// TIA Portal V17 export
// export: Created 2024-08-29T18:23:42.9804485Z, ExportSetting WithDefaults, DisplayName Totally Integrated Automation Portal, DisplayVersion V17 Update 7, DisplayName TIA Portal Openness, DisplayVersion V17 Update 7, DisplayName TIA Portal Version Control Interface, DisplayVersion V17, DisplayName SINAMICS Startdrive Advanced, DisplayVersion V17 SP2, DisplayName SINAMICS Startdrive G110M, G120, G120C, G120D, G120P, G115D, DisplayVersion V17 SP2, DisplayName SINAMICS Startdrive G130, G150, S120, S150, SINAMICS MV, S210, DisplayVersion V17 SP2, DisplayName STEP 7 Professional, DisplayVersion V17 Update 7, DisplayName STEP 7 Safety, DisplayVersion V17 Update 6, DisplayName WinCC Advanced / Unified PC, DisplayVersion V17 Update 7
FUNCTION "outputsMapping" : Void   // FC8, LAD
{ S7_Optimized_Access := 'TRUE' }
VERSION : 0.1
// stored: AutoNumber true, IsIECCheckEnabled false, SetENOAutomatically false, UDAEnableTagReadback false
BEGIN

REGION Network 1: STATION AIR ACTIVATION
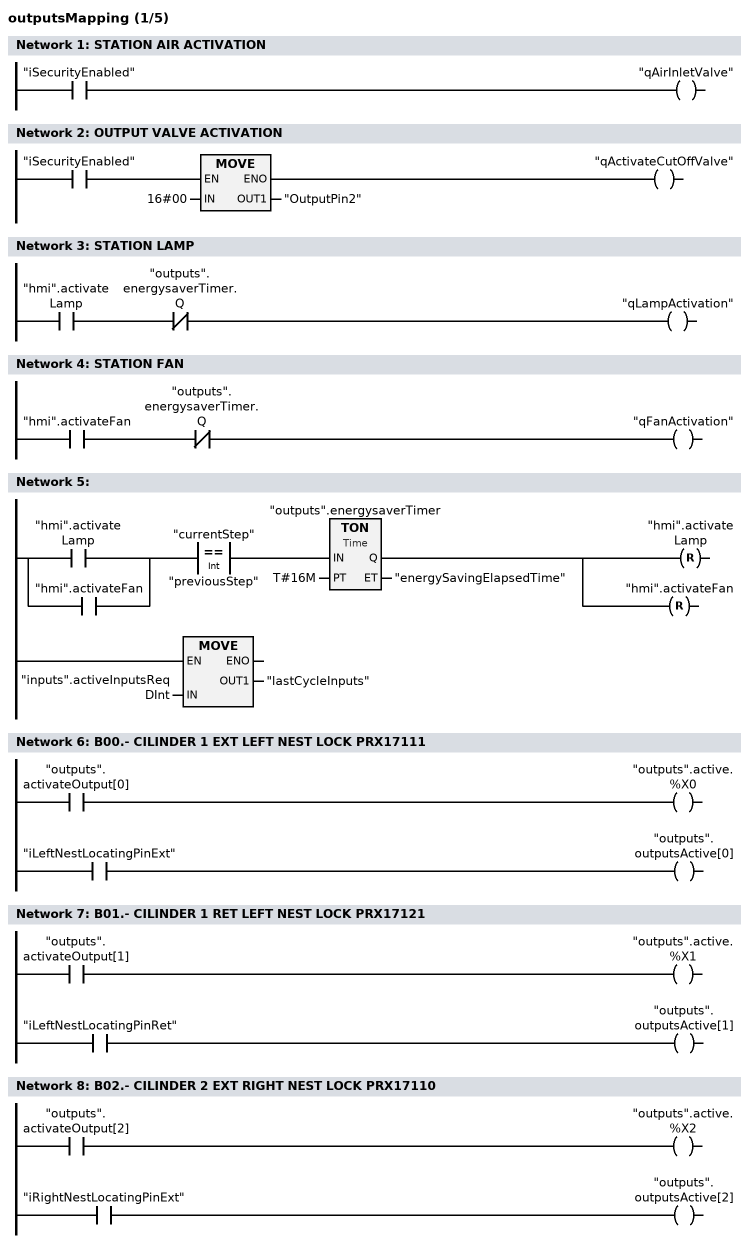
   RUNG wire#powerrail
      Contact( "iSecurityEnabled" )
      Coil( "qAirInletValve" )
   END_RUNG
   // the same network as SCL:
   "qAirInletValve" := "iSecurityEnabled";
END_REGION

REGION Network 2: OUTPUT VALVE ACTIVATION
   RUNG wire#powerrail
      Contact( "iSecurityEnabled" )
      Move(in := 16#00, out1 => "OutputPin2")
      Coil( "qActivateCutOffValve" )
   END_RUNG
   // the same network as SCL:
   IF "iSecurityEnabled" THEN "OutputPin2" := 16#00; END_IF;
   "qActivateCutOffValve" := "iSecurityEnabled";
END_REGION

REGION Network 3: STATION LAMP
   RUNG wire#powerrail
      Contact( "hmi".activateLamp )
      I_Contact( "outputs".energysaverTimer.Q )
      Coil( "qLampActivation" )
   END_RUNG
   // the same network as SCL:
   "qLampActivation" := "hmi".activateLamp AND NOT "outputs".energysaverTimer.Q;
END_REGION

REGION Network 4: STATION FAN
   RUNG wire#powerrail
      Contact( "hmi".activateFan )
      I_Contact( "outputs".energysaverTimer.Q )
      Coil( "qFanActivation" )
   END_RUNG
   // the same network as SCL:
   "qFanActivation" := "hmi".activateFan AND NOT "outputs".energysaverTimer.Q;
END_REGION

REGION Network 5
   RUNG wire#powerrail
      Contact( "hmi".activateLamp )
      wire#w1
      { S7_Templates := "SrcType := Int" } EQ_Contact(in1 := "currentStep", in2 := "previousStep")
      { S7_Templates := "time_type := Time" } "outputs".energysaverTimer.TON(pt := T#16M, et => "energySavingElapsedTime")
      wire#w2
      R_Coil( "hmi".activateLamp )
   END_RUNG
   RUNG wire#powerrail
      Contact( "hmi".activateFan )
   END_RUNG wire#w1
   RUNG wire#w2
      R_Coil( "hmi".activateFan )
   END_RUNG
   RUNG wire#powerrail
      Move(in := "inputs".activeInputsReqDInt, out1 => "lastCycleInputs")
   END_RUNG
   // the same network as SCL:
   "outputs".energysaverTimer.TON(IN := ("hmi".activateLamp OR "hmi".activateFan) AND ("currentStep" = "previousStep"),
                           PT := T#16M,
                           ET => "energySavingElapsedTime");
   IF "outputs".energysaverTimer.Q THEN
       "hmi".activateLamp := FALSE;
       "hmi".activateFan := FALSE;
   END_IF;
   "lastCycleInputs" := "inputs".activeInputsReqDInt;
END_REGION

REGION Network 6: B00.- CILINDER 1 EXT LEFT NEST LOCK PRX17111
   RUNG wire#powerrail
      Contact( "outputs".activateOutput[0] )
      Coil( "outputs".active.%X0 )
   END_RUNG
   RUNG wire#powerrail
      Contact( "iLeftNestLocatingPinExt" )
      Coil( "outputs".outputsActive[0] )
   END_RUNG
   // the same network as SCL:
   "outputs".active.%X0 := "outputs".activateOutput[0];
   "outputs".outputsActive[0] := "iLeftNestLocatingPinExt";
END_REGION

REGION Network 7: B01.- CILINDER 1 RET LEFT NEST LOCK PRX17121
   RUNG wire#powerrail
      Contact( "outputs".activateOutput[1] )
      Coil( "outputs".active.%X1 )
   END_RUNG
   RUNG wire#powerrail
      Contact( "iLeftNestLocatingPinRet" )
      Coil( "outputs".outputsActive[1] )
   END_RUNG
   // the same network as SCL:
   "outputs".active.%X1 := "outputs".activateOutput[1];
   "outputs".outputsActive[1] := "iLeftNestLocatingPinRet";
END_REGION

REGION Network 8: B02.- CILINDER 2 EXT RIGHT NEST LOCK PRX17110
   RUNG wire#powerrail
      Contact( "outputs".activateOutput[2] )
      Coil( "outputs".active.%X2 )
   END_RUNG
   RUNG wire#powerrail
      Contact( "iRightNestLocatingPinExt" )
      Coil( "outputs".outputsActive[2] )
   END_RUNG
   // the same network as SCL:
   "outputs".active.%X2 := "outputs".activateOutput[2];
   "outputs".outputsActive[2] := "iRightNestLocatingPinExt";
END_REGION

REGION Network 9: B03.- CILINDER 2 RET RIGHT NEST LOCK PRX17120
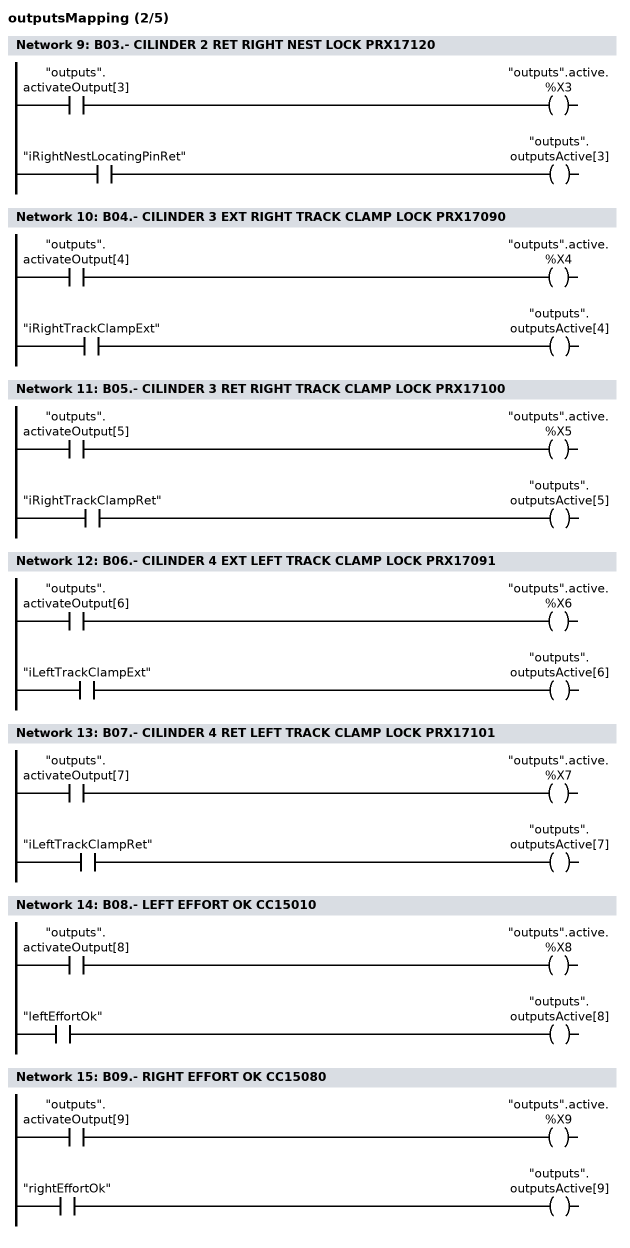
   RUNG wire#powerrail
      Contact( "outputs".activateOutput[3] )
      Coil( "outputs".active.%X3 )
   END_RUNG
   RUNG wire#powerrail
      Contact( "iRightNestLocatingPinRet" )
      Coil( "outputs".outputsActive[3] )
   END_RUNG
   // the same network as SCL:
   "outputs".active.%X3 := "outputs".activateOutput[3];
   "outputs".outputsActive[3] := "iRightNestLocatingPinRet";
END_REGION

REGION Network 10: B04.- CILINDER 3 EXT RIGHT TRACK CLAMP LOCK PRX17090
   RUNG wire#powerrail
      Contact( "outputs".activateOutput[4] )
      Coil( "outputs".active.%X4 )
   END_RUNG
   RUNG wire#powerrail
      Contact( "iRightTrackClampExt" )
      Coil( "outputs".outputsActive[4] )
   END_RUNG
   // the same network as SCL:
   "outputs".active.%X4 := "outputs".activateOutput[4];
   "outputs".outputsActive[4] := "iRightTrackClampExt";
END_REGION

REGION Network 11: B05.- CILINDER 3 RET RIGHT TRACK CLAMP LOCK PRX17100
   RUNG wire#powerrail
      Contact( "outputs".activateOutput[5] )
      Coil( "outputs".active.%X5 )
   END_RUNG
   RUNG wire#powerrail
      Contact( "iRightTrackClampRet" )
      Coil( "outputs".outputsActive[5] )
   END_RUNG
   // the same network as SCL:
   "outputs".active.%X5 := "outputs".activateOutput[5];
   "outputs".outputsActive[5] := "iRightTrackClampRet";
END_REGION

REGION Network 12: B06.- CILINDER 4 EXT LEFT TRACK CLAMP LOCK PRX17091
   RUNG wire#powerrail
      Contact( "outputs".activateOutput[6] )
      Coil( "outputs".active.%X6 )
   END_RUNG
   RUNG wire#powerrail
      Contact( "iLeftTrackClampExt" )
      Coil( "outputs".outputsActive[6] )
   END_RUNG
   // the same network as SCL:
   "outputs".active.%X6 := "outputs".activateOutput[6];
   "outputs".outputsActive[6] := "iLeftTrackClampExt";
END_REGION

REGION Network 13: B07.- CILINDER 4 RET LEFT TRACK CLAMP LOCK PRX17101
   RUNG wire#powerrail
      Contact( "outputs".activateOutput[7] )
      Coil( "outputs".active.%X7 )
   END_RUNG
   RUNG wire#powerrail
      Contact( "iLeftTrackClampRet" )
      Coil( "outputs".outputsActive[7] )
   END_RUNG
   // the same network as SCL:
   "outputs".active.%X7 := "outputs".activateOutput[7];
   "outputs".outputsActive[7] := "iLeftTrackClampRet";
END_REGION

REGION Network 14: B08.- LEFT EFFORT OK CC15010
   RUNG wire#powerrail
      Contact( "outputs".activateOutput[8] )
      Coil( "outputs".active.%X8 )
   END_RUNG
   RUNG wire#powerrail
      Contact( "leftEffortOk" )
      Coil( "outputs".outputsActive[8] )
   END_RUNG
   // the same network as SCL:
   "outputs".active.%X8 := "outputs".activateOutput[8];
   "outputs".outputsActive[8] := "leftEffortOk";
END_REGION

REGION Network 15: B09.- RIGHT EFFORT OK CC15080
   RUNG wire#powerrail
      Contact( "outputs".activateOutput[9] )
      Coil( "outputs".active.%X9 )
   END_RUNG
   RUNG wire#powerrail
      Contact( "rightEffortOk" )
      Coil( "outputs".outputsActive[9] )
   END_RUNG
   // the same network as SCL:
   "outputs".active.%X9 := "outputs".activateOutput[9];
   "outputs".outputsActive[9] := "rightEffortOk";
END_REGION

REGION Network 16: B10.- LEFT INSERTION OK DISTANCE SD14160
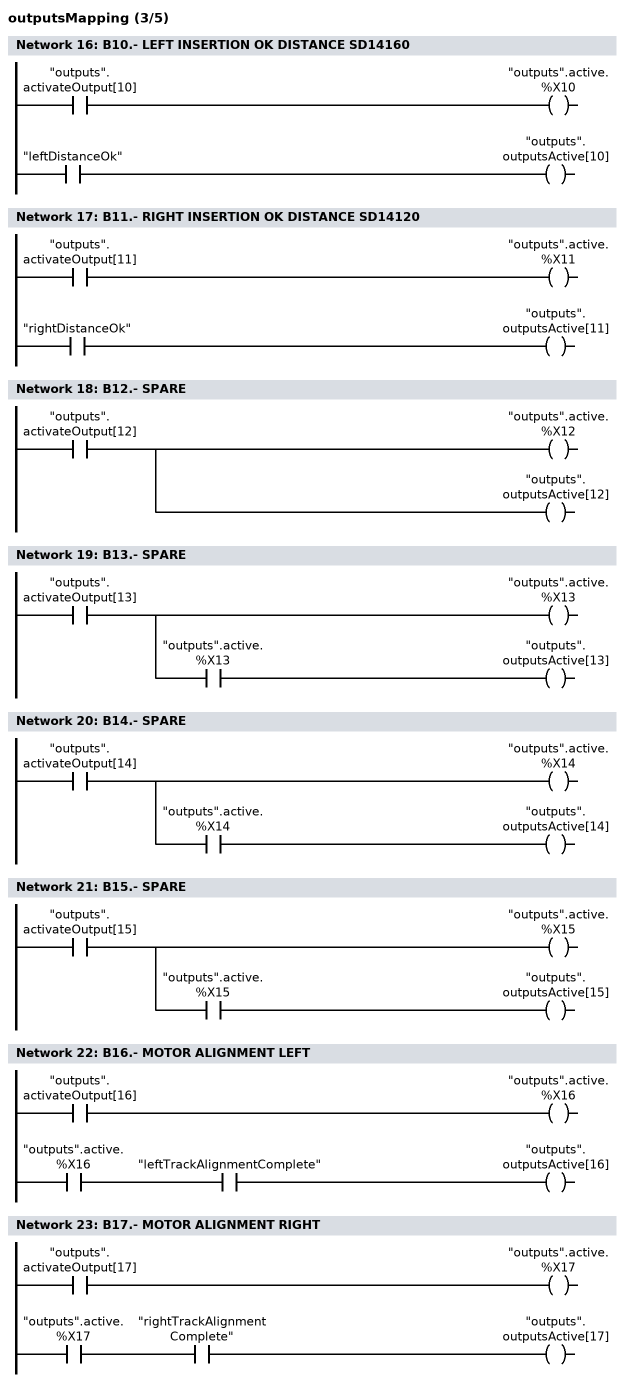
   RUNG wire#powerrail
      Contact( "outputs".activateOutput[10] )
      Coil( "outputs".active.%X10 )
   END_RUNG
   RUNG wire#powerrail
      Contact( "leftDistanceOk" )
      Coil( "outputs".outputsActive[10] )
   END_RUNG
   // the same network as SCL:
   "outputs".active.%X10 := "outputs".activateOutput[10];
   "outputs".outputsActive[10] := "leftDistanceOk";
END_REGION

REGION Network 17: B11.- RIGHT INSERTION OK DISTANCE SD14120
   RUNG wire#powerrail
      Contact( "outputs".activateOutput[11] )
      Coil( "outputs".active.%X11 )
   END_RUNG
   RUNG wire#powerrail
      Contact( "rightDistanceOk" )
      Coil( "outputs".outputsActive[11] )
   END_RUNG
   // the same network as SCL:
   "outputs".active.%X11 := "outputs".activateOutput[11];
   "outputs".outputsActive[11] := "rightDistanceOk";
END_REGION

REGION Network 18: B12.- SPARE
   RUNG wire#powerrail
      Contact( "outputs".activateOutput[12] )
      wire#w1
      Coil( "outputs".active.%X12 )
   END_RUNG
   RUNG wire#w1
      Coil( "outputs".outputsActive[12] )
   END_RUNG
   // the same network as SCL:
   "outputs".active.%X12 := "outputs".activateOutput[12];
   "outputs".outputsActive[12] := "outputs".activateOutput[12];
END_REGION

REGION Network 19: B13.- SPARE
   RUNG wire#powerrail
      Contact( "outputs".activateOutput[13] )
      wire#w1
      Coil( "outputs".active.%X13 )
   END_RUNG
   RUNG wire#w1
      Contact( "outputs".active.%X13 )
      Coil( "outputs".outputsActive[13] )
   END_RUNG
   // the same network as SCL:
   "outputs".active.%X13 := "outputs".activateOutput[13];
   "outputs".outputsActive[13] := "outputs".activateOutput[13] AND "outputs".active.%X13;
END_REGION

REGION Network 20: B14.- SPARE
   RUNG wire#powerrail
      Contact( "outputs".activateOutput[14] )
      wire#w1
      Coil( "outputs".active.%X14 )
   END_RUNG
   RUNG wire#w1
      Contact( "outputs".active.%X14 )
      Coil( "outputs".outputsActive[14] )
   END_RUNG
   // the same network as SCL:
   "outputs".active.%X14 := "outputs".activateOutput[14];
   "outputs".outputsActive[14] := "outputs".activateOutput[14] AND "outputs".active.%X14;
END_REGION

REGION Network 21: B15.- SPARE
   RUNG wire#powerrail
      Contact( "outputs".activateOutput[15] )
      wire#w1
      Coil( "outputs".active.%X15 )
   END_RUNG
   RUNG wire#w1
      Contact( "outputs".active.%X15 )
      Coil( "outputs".outputsActive[15] )
   END_RUNG
   // the same network as SCL:
   "outputs".active.%X15 := "outputs".activateOutput[15];
   "outputs".outputsActive[15] := "outputs".activateOutput[15] AND "outputs".active.%X15;
END_REGION

REGION Network 22: B16.- MOTOR ALIGNMENT LEFT
   RUNG wire#powerrail
      Contact( "outputs".activateOutput[16] )
      Coil( "outputs".active.%X16 )
   END_RUNG
   RUNG wire#powerrail
      Contact( "outputs".active.%X16 )
      Contact( "leftTrackAlignmentComplete" )
      Coil( "outputs".outputsActive[16] )
   END_RUNG
   // the same network as SCL:
   "outputs".active.%X16 := "outputs".activateOutput[16];
   "outputs".outputsActive[16] := "outputs".active.%X16 AND "leftTrackAlignmentComplete";
END_REGION

REGION Network 23: B17.- MOTOR ALIGNMENT RIGHT
   RUNG wire#powerrail
      Contact( "outputs".activateOutput[17] )
      Coil( "outputs".active.%X17 )
   END_RUNG
   RUNG wire#powerrail
      Contact( "outputs".active.%X17 )
      Contact( "rightTrackAlignmentComplete" )
      Coil( "outputs".outputsActive[17] )
   END_RUNG
   // the same network as SCL:
   "outputs".active.%X17 := "outputs".activateOutput[17];
   "outputs".outputsActive[17] := "outputs".active.%X17 AND "rightTrackAlignmentComplete";
END_REGION

REGION Network 24: B18.- SPARE
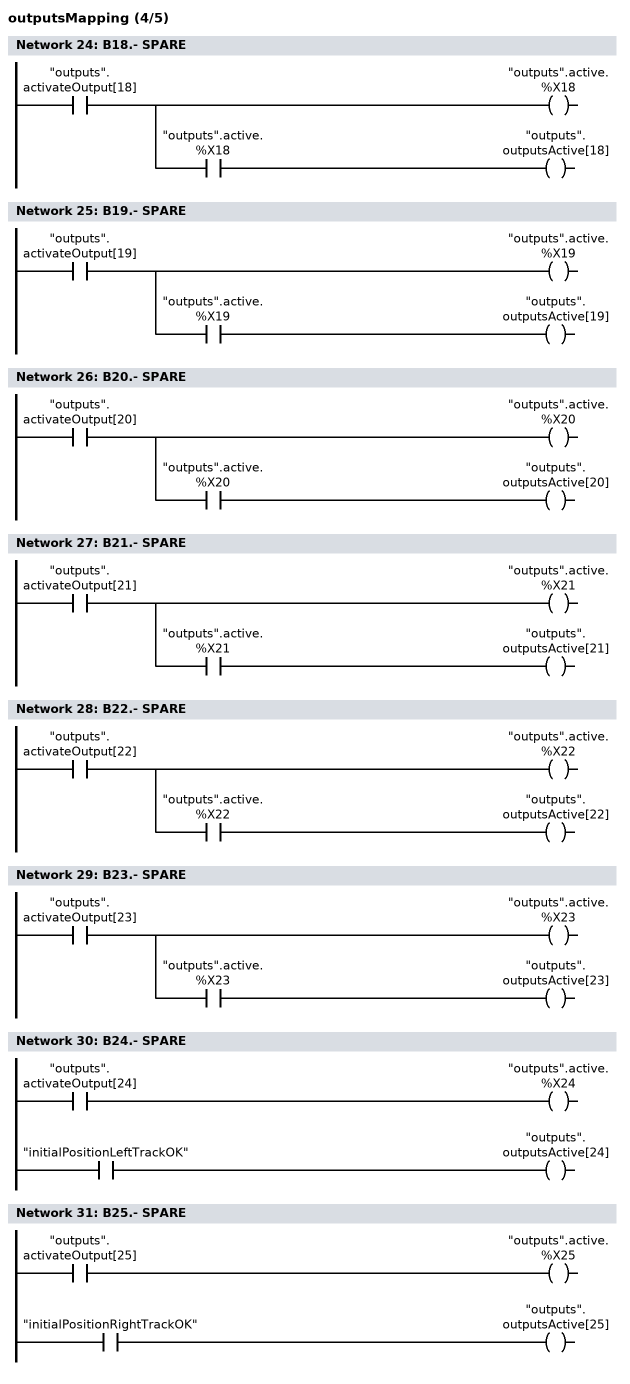
   RUNG wire#powerrail
      Contact( "outputs".activateOutput[18] )
      wire#w1
      Coil( "outputs".active.%X18 )
   END_RUNG
   RUNG wire#w1
      Contact( "outputs".active.%X18 )
      Coil( "outputs".outputsActive[18] )
   END_RUNG
   // the same network as SCL:
   "outputs".active.%X18 := "outputs".activateOutput[18];
   "outputs".outputsActive[18] := "outputs".activateOutput[18] AND "outputs".active.%X18;
END_REGION

REGION Network 25: B19.- SPARE
   RUNG wire#powerrail
      Contact( "outputs".activateOutput[19] )
      wire#w1
      Coil( "outputs".active.%X19 )
   END_RUNG
   RUNG wire#w1
      Contact( "outputs".active.%X19 )
      Coil( "outputs".outputsActive[19] )
   END_RUNG
   // the same network as SCL:
   "outputs".active.%X19 := "outputs".activateOutput[19];
   "outputs".outputsActive[19] := "outputs".activateOutput[19] AND "outputs".active.%X19;
END_REGION

REGION Network 26: B20.- SPARE
   RUNG wire#powerrail
      Contact( "outputs".activateOutput[20] )
      wire#w1
      Coil( "outputs".active.%X20 )
   END_RUNG
   RUNG wire#w1
      Contact( "outputs".active.%X20 )
      Coil( "outputs".outputsActive[20] )
   END_RUNG
   // the same network as SCL:
   "outputs".active.%X20 := "outputs".activateOutput[20];
   "outputs".outputsActive[20] := "outputs".activateOutput[20] AND "outputs".active.%X20;
END_REGION

REGION Network 27: B21.- SPARE
   RUNG wire#powerrail
      Contact( "outputs".activateOutput[21] )
      wire#w1
      Coil( "outputs".active.%X21 )
   END_RUNG
   RUNG wire#w1
      Contact( "outputs".active.%X21 )
      Coil( "outputs".outputsActive[21] )
   END_RUNG
   // the same network as SCL:
   "outputs".active.%X21 := "outputs".activateOutput[21];
   "outputs".outputsActive[21] := "outputs".activateOutput[21] AND "outputs".active.%X21;
END_REGION

REGION Network 28: B22.- SPARE
   RUNG wire#powerrail
      Contact( "outputs".activateOutput[22] )
      wire#w1
      Coil( "outputs".active.%X22 )
   END_RUNG
   RUNG wire#w1
      Contact( "outputs".active.%X22 )
      Coil( "outputs".outputsActive[22] )
   END_RUNG
   // the same network as SCL:
   "outputs".active.%X22 := "outputs".activateOutput[22];
   "outputs".outputsActive[22] := "outputs".activateOutput[22] AND "outputs".active.%X22;
END_REGION

REGION Network 29: B23.- SPARE
   RUNG wire#powerrail
      Contact( "outputs".activateOutput[23] )
      wire#w1
      Coil( "outputs".active.%X23 )
   END_RUNG
   RUNG wire#w1
      Contact( "outputs".active.%X23 )
      Coil( "outputs".outputsActive[23] )
   END_RUNG
   // the same network as SCL:
   "outputs".active.%X23 := "outputs".activateOutput[23];
   "outputs".outputsActive[23] := "outputs".activateOutput[23] AND "outputs".active.%X23;
END_REGION

REGION Network 30: B24.- SPARE
   RUNG wire#powerrail
      Contact( "outputs".activateOutput[24] )
      Coil( "outputs".active.%X24 )
   END_RUNG
   RUNG wire#powerrail
      Contact( "initialPositionLeftTrackOK" )
      Coil( "outputs".outputsActive[24] )
   END_RUNG
   // the same network as SCL:
   "outputs".active.%X24 := "outputs".activateOutput[24];
   "outputs".outputsActive[24] := "initialPositionLeftTrackOK";
END_REGION

REGION Network 31: B25.- SPARE
   RUNG wire#powerrail
      Contact( "outputs".activateOutput[25] )
      Coil( "outputs".active.%X25 )
   END_RUNG
   RUNG wire#powerrail
      Contact( "initialPositionRightTrackOK" )
      Coil( "outputs".outputsActive[25] )
   END_RUNG
   // the same network as SCL:
   "outputs".active.%X25 := "outputs".activateOutput[25];
   "outputs".outputsActive[25] := "initialPositionRightTrackOK";
END_REGION

REGION Network 32: B26.- SPARE
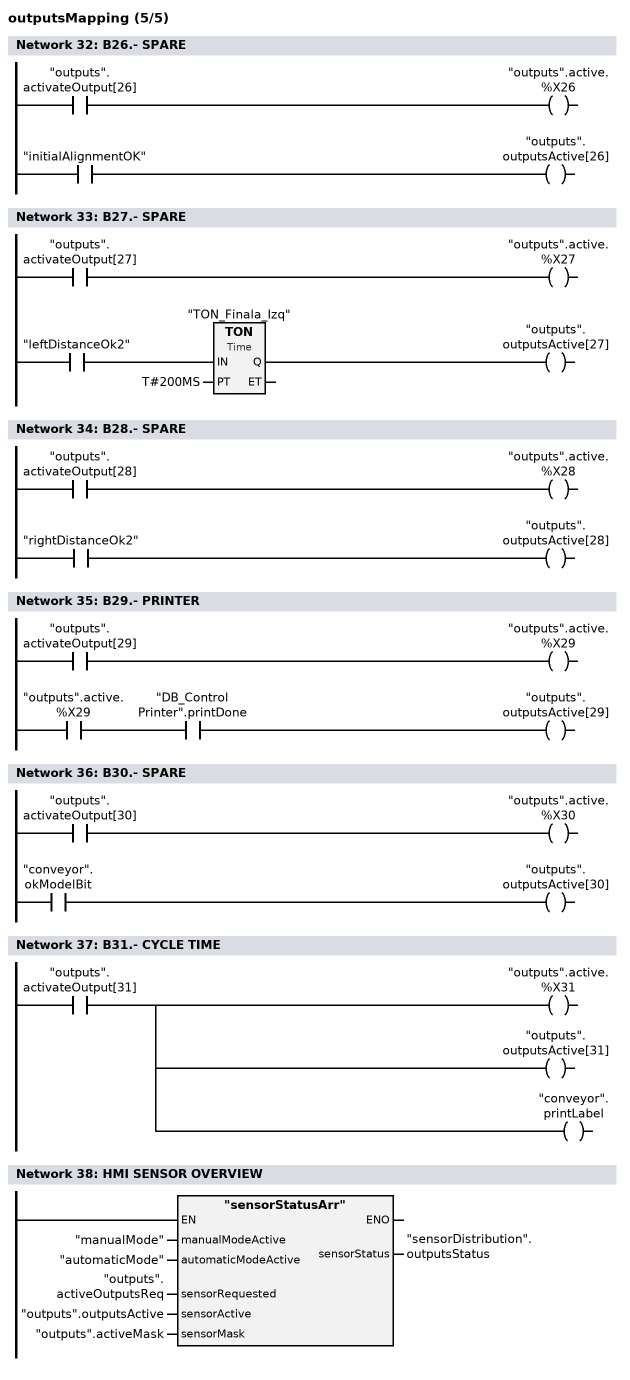
   RUNG wire#powerrail
      Contact( "outputs".activateOutput[26] )
      Coil( "outputs".active.%X26 )
   END_RUNG
   RUNG wire#powerrail
      Contact( "initialAlignmentOK" )
      Coil( "outputs".outputsActive[26] )
   END_RUNG
   // the same network as SCL:
   "outputs".active.%X26 := "outputs".activateOutput[26];
   "outputs".outputsActive[26] := "initialAlignmentOK";
END_REGION

REGION Network 33: B27.- SPARE
   RUNG wire#powerrail
      Contact( "outputs".activateOutput[27] )
      Coil( "outputs".active.%X27 )
   END_RUNG
   RUNG wire#powerrail
      Contact( "leftDistanceOk2" )
      { S7_Templates := "time_type := Time" } "TON_Finala_Izq".TON(pt := T#200MS, et =>)
      Coil( "outputs".outputsActive[27] )
   END_RUNG
   // the same network as SCL:
   "outputs".active.%X27 := "outputs".activateOutput[27];
   "TON_Finala_Izq".TON(IN := "leftDistanceOk2", PT := T#200MS);
   "outputs".outputsActive[27] := "TON_Finala_Izq".Q;
END_REGION

REGION Network 34: B28.- SPARE
   RUNG wire#powerrail
      Contact( "outputs".activateOutput[28] )
      Coil( "outputs".active.%X28 )
   END_RUNG
   RUNG wire#powerrail
      Contact( "rightDistanceOk2" )
      Coil( "outputs".outputsActive[28] )
   END_RUNG
   // the same network as SCL:
   "outputs".active.%X28 := "outputs".activateOutput[28];
   "outputs".outputsActive[28] := "rightDistanceOk2";
END_REGION

REGION Network 35: B29.- PRINTER
   RUNG wire#powerrail
      Contact( "outputs".activateOutput[29] )
      Coil( "outputs".active.%X29 )
   END_RUNG
   RUNG wire#powerrail
      Contact( "outputs".active.%X29 )
      Contact( "DB_ControlPrinter".printDone )
      Coil( "outputs".outputsActive[29] )
   END_RUNG
   // the same network as SCL:
   "outputs".active.%X29 := "outputs".activateOutput[29];
   "outputs".outputsActive[29] := "outputs".active.%X29 AND "DB_ControlPrinter".printDone;
END_REGION

REGION Network 36: B30.- SPARE
   RUNG wire#powerrail
      Contact( "outputs".activateOutput[30] )
      Coil( "outputs".active.%X30 )
   END_RUNG
   RUNG wire#powerrail
      Contact( "conveyor".okModelBit )
      Coil( "outputs".outputsActive[30] )
   END_RUNG
   // the same network as SCL:
   "outputs".active.%X30 := "outputs".activateOutput[30];
   "outputs".outputsActive[30] := "conveyor".okModelBit;
END_REGION

REGION Network 37: B31.- CYCLE TIME
   RUNG wire#powerrail
      Contact( "outputs".activateOutput[31] )
      wire#w1
      Coil( "outputs".active.%X31 )
   END_RUNG
   RUNG wire#w1
      Coil( "outputs".outputsActive[31] )
   END_RUNG
   RUNG wire#w1
      Coil( "conveyor".printLabel )
   END_RUNG
   // the same network as SCL:
   "outputs".active.%X31 := "outputs".activateOutput[31];
   "outputs".outputsActive[31] := "outputs".activateOutput[31];
   "conveyor".printLabel := "outputs".activateOutput[31];
END_REGION

REGION Network 38: HMI SENSOR OVERVIEW
   RUNG wire#powerrail
      "sensorStatusArr"(manualModeActive := "manualMode", automaticModeActive := "automaticMode", sensorRequested := "outputs".activeOutputsReq, sensorActive := "outputs".outputsActive, sensorMask := "outputs".activeMask, sensorStatus => "sensorDistribution".outputsStatus)
   END_RUNG
   // the same network as SCL:
   "sensorStatusArr"(manualModeActive := "manualMode",
                     automaticModeActive := "automaticMode",
                     sensorRequested := "outputs".activeOutputsReq,
                     sensorActive := "outputs".outputsActive,
                     sensorMask := "outputs".activeMask,
                     sensorStatus => "sensorDistribution".outputsStatus);
END_REGION
END_FUNCTION
